Fanuc KAREL source: kt00890.KL

-- PROVISIONAL review KL for V770-1; original PC SHA256 58f7ca88f62eebb0c107892e26fb7c6bbf35cc692549d28b2e2eef2790017426
-- Incomplete behavior may be omitted. Consult companion uncertainty JSON. Do not deploy.
PROGRAM KT00890
%NOLOCKGROUP
-- UNRESOLVED_DECL P1 type=000106
-- UNRESOLVED_DECL P2 type=000106
-- UNRESOLVED_DECL OUT type=000101
BEGIN
  -- UNRESOLVED_PC offsets 5-20; opcodes 2E,22,32,35
  -- UNRESOLVED_PC offsets 25-40; opcodes 2E,22,32,35
  -- UNRESOLVED_PC offsets 45-60; opcodes 2E,22,32,35
  -- UNRESOLVED_PC offsets 65-80; opcodes 2E,22,32,35
  -- UNRESOLVED_PC offsets 85-115; opcodes 27,27,49,7E,AD,76,7E,4A
  -- UNRESOLVED_PC offsets 120-124; opcodes 7F
END KT00890
